// TIA Portal V17 export
// export: Created 2024-10-17T14:16:15.9801072Z, ExportSetting WithDefaults, DisplayName Totally Integrated Automation Portal, DisplayVersion V17 Update 4, DisplayName TIA Portal Openness, DisplayVersion V17 Update 4, DisplayName TIA Portal Version Control Interface, DisplayVersion V17, DisplayName SINAMICS Startdrive Advanced, DisplayVersion V17 Update2, DisplayName SINAMICS Startdrive G130, G150, S120, S150, SINAMICS MV, S210, DisplayVersion V17 Update2, DisplayName SINAMICS Startdrive G110M, G120, G120C, G120D, G120P, G115D, DisplayVersion V17 Update2, DisplayName STEP 7 Professional, DisplayVersion V17 Update 4, DisplayName STEP 7 Safety, DisplayVersion V17, DisplayName WinCC Advanced / Unified PC, DisplayVersion V17 Update 4
DATA_BLOCK "PACKMLV2022"   // DB30135
TITLE = PackTags DB
{ S7_Optimized_Access := 'TRUE' }
VERSION : 0.1
// stored: AutoNumber true, DBAccessibleFromOPCUA true, DBAccessibleFromWebserver true, InstanceOfName LPMLV2022_typePackTags, InstanceOfType UDT, IsOnlyStoredInLoadMemory false, IsWriteProtectedInAS false
"LPMLV2022_typePackTags"
   // VAR
   //    Command : "LPMLV2022_typeCommand";
   //    Status { ExternalWritable := 'False'} : "LPMLV2022_typeStatus";
   //    Admin { ExternalWritable := 'False'} : "LPMLV2022_typeAdmin";
   // END_VAR
BEGIN
END_DATA_BLOCK
